// Mitsubishi GX Works2 project: Rev   PLC: Q00J

PROGRAM MAIN
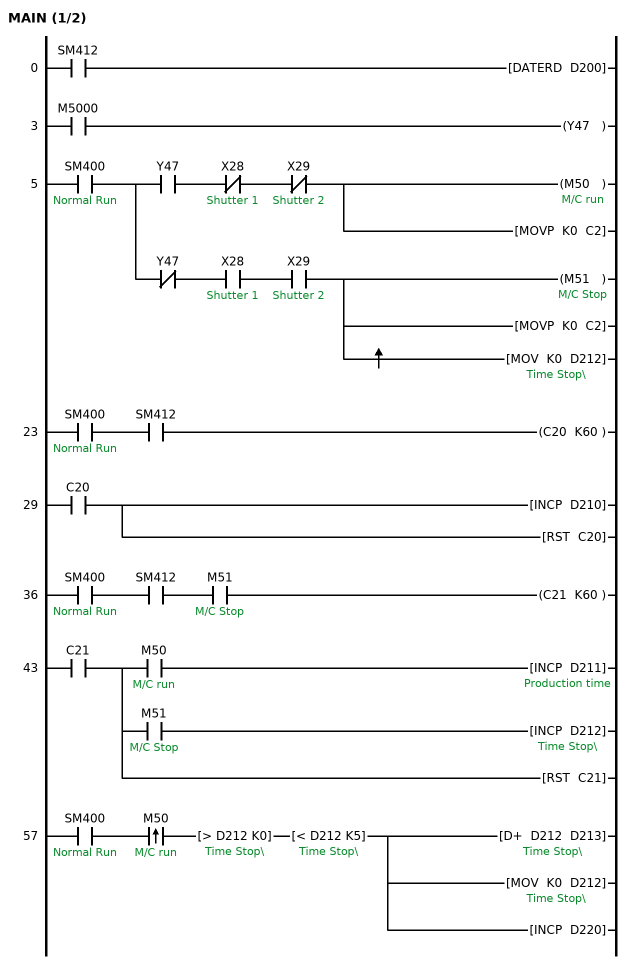
0     LD      SM412
      DATERD  D200
3     LD      M5000
      OUT     Y47
5     LD      SM400  ; Normal Run
      MPS
      AND     Y47
      ANI     X28  ; Shutter 1
      ANI     X29  ; Shutter 2
      OUT     M50  ; M/C run
      MOVP    K0 C2
      MPP
      ANI     Y47
      AND     X28  ; Shutter 1
      AND     X29  ; Shutter 2
      OUT     M51  ; M/C Stop
      MOVP    K0 C2
      MEP
      MOV     K0 D212  ; Time Stop\
23    LD      SM400  ; Normal Run
      AND     SM412
      OUT     C20 K60
29    LD      C20
      INCP    D210
      RST     C20
36    LD      SM400  ; Normal Run
      AND     SM412
      AND     M51  ; M/C Stop
      OUT     C21 K60
43    LD      C21
      MPS
      AND     M50  ; M/C run
      INCP    D211  ; Production time
      MRD
      AND     M51  ; M/C Stop
      INCP    D212
      MPP
      RST     C21
57    LD      SM400  ; Normal Run
      ANDP    M50  ; M/C run
      AND>    D212 K0  ; Time Stop\
      AND<    D212 K5  ; Time Stop\
      D+      D212 D213
      MOV     K0 D212
      INCP    D220
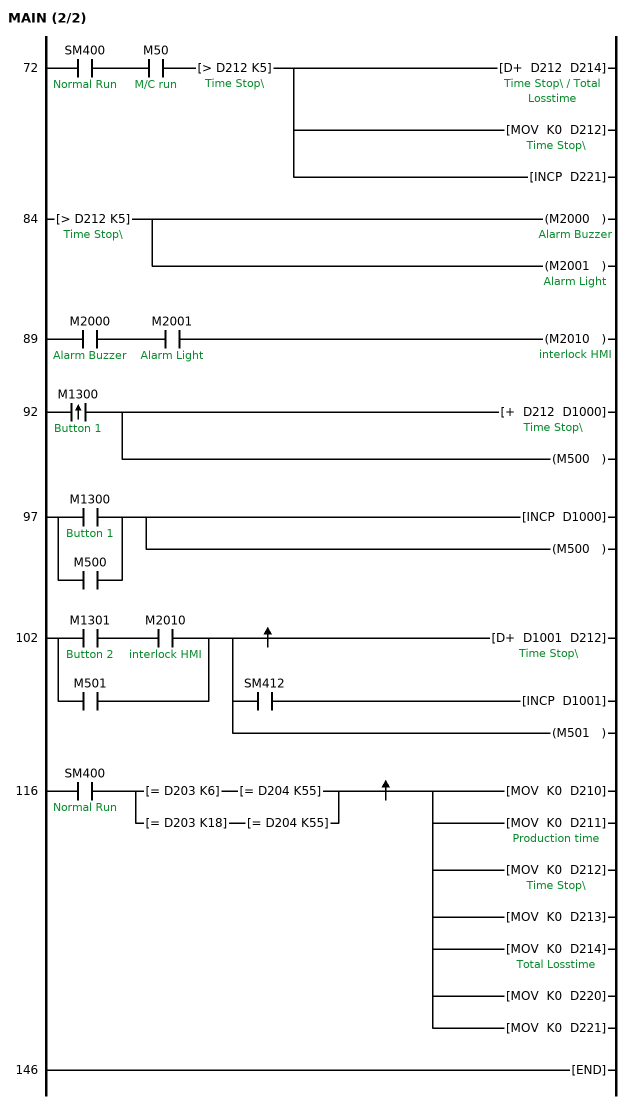
72    LD      SM400  ; Normal Run
      AND     M50  ; M/C run
      AND>    D212 K5  ; Time Stop\
      D+      D212 D214  ; Total Losstime
      MOV     K0 D212
      INCP    D221
84    LD>     D212 K5  ; Time Stop\
      OUT     M2000  ; Alarm Buzzer
      OUT     M2001  ; Alarm Light
89    LD      M2000  ; Alarm Buzzer
      AND     M2001  ; Alarm Light
      OUT     M2010  ; interlock HMI
92    LDP     M1300  ; Button 1
      +       D212 D1000
      OUT     M500
97    LD      M1300  ; Button 1
      OR      M500
      INCP    D1000
      OUT     M500
102   LD      M1301  ; Button 2
      AND     M2010  ; interlock HMI
      OR      M501
      MPS
      MEP
      D+      D1001 D212
      MRD
      AND     SM412
      INCP    D1001
      MPP
      OUT     M501
116   LD      SM400  ; Normal Run
      LD=     D203 K6
      AND=    D204 K55
      LD=     D203 K18
      AND=    D204 K55
      ORB
      ANB
      MEP
      MOV     K0 D210
      MOV     K0 D211
      MOV     K0 D212
      MOV     K0 D213
      MOV     K0 D214
      MOV     K0 D220
      MOV     K0 D221
146   END
END_PROGRAM
